FUNCTION_BLOCK E_T_FF (* Toggle flip flop *)
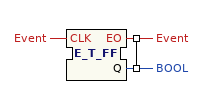
  EVENT_INPUT
    CLK; (* Clock for triggering a output toggle *)
  END_EVENT
  EVENT_OUTPUT
    EO WITH Q; (* Output Q has changed *)
  END_EVENT
  VAR_OUTPUT
    Q : BOOL; (* value of flip flop *)
  END_VAR
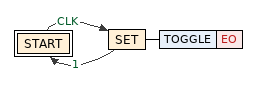
  EC_STATES
    START; (* Initial State *)
    SET : TOGGLE -> EO; (* Initialization *)
  END_STATES
  EC_TRANSITIONS
    START TO SET := CLK;
    SET TO START := 1;
  END_TRANSITIONS
  ALGORITHM TOGGLE IN ST: (* TOGGLE algorithm *)
Q := NOT Q;
  END_ALGORITHM
END_FUNCTION_BLOCK
